FUNCTION_BLOCK AI_FB_CTD (* Down counter (INT) AI-Adapter Version *)
  (* Standard: 61499-2; Description: Copyright (c) 2026 Meisterschulen am Ostbahnhof This program and the accompanying materials are made available under the terms of the Eclipse Public License 2.0 which is available at https://www.eclipse.org/legal/epl-2.0/ SPDX-License-Identifier: EPL-2.0 NOTE: This block fires the AX output event (Q.E1) on every update (CD, LD, PV). If on-change triggering is required, use of an AX_D_FF as a filter is recommended. *)
  (* Version 1.0, 2026-04-21, Franz Höpfinger, Meisterschulen am Ostbahnhof, initial API and implementation and/or initial documentation *)
  PACKAGE adapter::iec61131_3::counters;
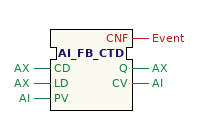
  EVENT_OUTPUT
    CNF; (* Execution Confirmation *)
  END_EVENT
  SOCKETS
    CD : adapter::types::unidirectional::AX; (* Count down *)
    LD : adapter::types::unidirectional::AX; (* Load *)
    PV : adapter::types::unidirectional::AI; (* Preset value *)
  END_SOCKETS
  PLUGS
    Q : adapter::types::unidirectional::AX; (* Output *)
    CV : adapter::types::unidirectional::AI; (* Count value *)
  END_PLUGS
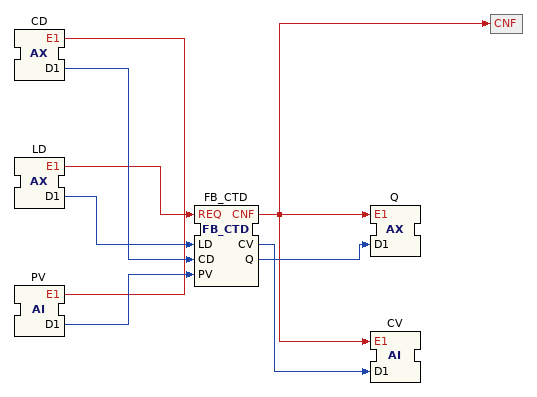
  FBS
    FB_CTD : iec61131::counters::FB_CTD;
  END_FBS
  EVENT_CONNECTIONS
    LD.E1 TO FB_CTD.REQ;
    CD.E1 TO FB_CTD.REQ;
    PV.E1 TO FB_CTD.REQ;
    FB_CTD.CNF TO CV.E1;
    FB_CTD.CNF TO Q.E1;
    FB_CTD.CNF TO CNF;
  END_CONNECTIONS
  DATA_CONNECTIONS
    LD.D1 TO FB_CTD.LD;
    CD.D1 TO FB_CTD.CD;
    PV.D1 TO FB_CTD.PV;
    FB_CTD.CV TO CV.D1;
    FB_CTD.Q TO Q.D1;
  END_CONNECTIONS
END_FUNCTION_BLOCK
